FUNCTION_BLOCK NormallyClosePushButton IMPLEMENTS I_PushButton
VAR
	input AT%I* : BOOL;
END_VAR

PROPERTY PUBLIC isPressed : BOOL
GET
isPressed	:=	NOT input;
END_GET
END_PROPERTY

PROPERTY PUBLIC isReleased : BOOL
GET
isReleased	:=	input;
END_GET
END_PROPERTY

END_FUNCTION_BLOCK

(* stored: Version 1.1.0.1, ProductVersion 3.1.4024.12
   POU NormallyClosePushButton: Id {81f79b6c-6478-4cc2-9179-24a5b6aa895f}, SpecialFunc None
   Property isPressed: Id {ddf9cd05-5ad4-42e1-84cc-e3d3846bafcf}
   Get Get: Id {82c3a84a-9060-4e4e-90ed-7c9f0015d925}
   Property isReleased: Id {4fda6a0e-42df-4db9-b30c-e24295e3562d}
   Get Get: Id {e187bf4f-eb66-4c38-8b2a-d3cfb1c4a8c3} *)
